FUNCTION_BLOCK ABSTRACT FB_Axis_HomeToHardStop EXTENDS FB_AxisBase
VAR_INPUT
END_VAR
VAR_OUTPUT
END_VAR
VAR
	//Internal Property Variables
	fHomePositionSetpoint		: LREAL := 0;
	nTorqueLimit				: LREAL := 20;
	nTorqueFeedback				: DINT;
	eHomeDirection				: Tc2_MC2.MC_Direction := Tc2_MC2.MC_Direction.MC_Positive_Direction;
	
	//Misc
	a_AverageForceArray			: ARRAY[0..9] OF LREAL;
	i							: UINT;
	fDriveForce					: LREAL;
	fActualForce				: LREAL;
	fAverageForce				: LREAL;
END_VAR

PROPERTY AverageForce : LREAL
GET
AverageForce := fAverageForce;
END_GET
END_PROPERTY

PROPERTY HomeDirection : Tc2_MC2.MC_Direction
GET
HomeDirection := eHomeDirection;
END_GET
SET
eHomeDirection := HomeDirection;
END_SET
END_PROPERTY

PROPERTY HomePositionSetpoint : LREAL
GET
HomePositionSetpoint := fHomePositionSetpoint;
END_GET
SET
fHomePositionSetpoint := HomePositionSetpoint;
END_SET
END_PROPERTY

METHOD MotionControl : BOOL
VAR_INPUT
END_VAR
SUPER^.MotionControl();

//TODO: Set Torque Limit := LREAL_TO_INT(nTorqueLimit/0.051);

fActualForce := DINT_TO_INT(nTorqueFeedback)/10.0;

fAverageForce := fActualForce / 10;
FOR i := 9 TO 1 BY -1 DO
	a_AverageForceArray[i] := a_AverageForceArray[i-1];
	fAverageForce := fAverageForce + a_AverageForceArray[i]/10;
END_FOR
a_AverageForceArray[0] := fActualForce;

fbAxisHome.Options.SearchDirection := eHomeDirection;
fbAxisHome.Options.SearchVelocity := 2;
//Performs a simple home-to sensor sequence when commanded by a "Home" Method call
fbAxisHome(
	Axis:= SelectedAxis,
	Position:= fHomePositionSetpoint, 
	HomingMode:= MC_HomingMode.MC_DefaultHoming, 
	BufferMode:= MC_BufferMode.MC_Aborting,
	bCalibrationCam := ABS(fAverageForce) > ABS(nTorqueLimit));

fbAxisHome.Execute := FALSE;
END_METHOD

PROPERTY TorqueFeedback : DINT //1000 = 100%
GET
TorqueFeedback := nTorqueFeedback;
END_GET
END_PROPERTY

PROPERTY TorqueLimit : LREAL //1000 = 100%
GET
TorqueLimit := nTorqueLimit;
END_GET
SET
nTorqueLimit := TorqueLimit;
END_SET
END_PROPERTY

END_FUNCTION_BLOCK

(* stored: Version 1.1.0.1, ProductVersion 3.1.4024.9
   POU FB_Axis_HomeToHardStop: Id {ee534ea3-5ccb-48b7-bdbb-c927a5a91b95}, SpecialFunc None
   Folder 01_SUPER_Overrides: Id {b619ec89-4554-4ed7-b36c-4ce55535be3c}
   Property AverageForce: Id {38a9cc8c-621e-4418-9ccc-b99aefecd122}
   Get Get: Id {332b6257-a84b-4c3b-87f0-d448929f2126}
   Property HomeDirection: Id {144ce852-bcb6-4576-b7b7-9fadee241544}
   Get Get: Id {d602bcdc-ae47-4702-a64b-20f75afb79c8}
   Set Set: Id {6c99cbed-0c0d-445b-b25a-0fb5db5b2b22}
   Property HomePositionSetpoint: Id {30a0d12c-1f70-4239-b2d6-57812229cc91}
   Get Get: Id {8be4af57-74d6-43ab-9907-42896ce9dc25}
   Set Set: Id {457b453e-ebf0-44ad-9637-f09f9fa81106}
   Method MotionControl: Id {5202ea77-8ac8-41e4-aff3-c26d70b34fd9}
   Property TorqueFeedback: Id {c48650fe-6598-41e6-8e37-640e44978175}
   Get Get: Id {1de39173-b871-49eb-8cf6-cf69f98812b2}
   Property TorqueLimit: Id {3e887d3f-410c-4428-9059-52e5d771a8d2}
   Get Get: Id {6beca81e-5c94-4e9b-b1fd-38eafa9d6365}
   Set Set: Id {1e4f6015-7fbf-490f-ba28-e5199afee31d} *)
